// TIA Portal V19 export
ORGANIZATION_BLOCK "Main"   // OB3101, LAD, ProgramCycle
TITLE = "Main Program Sweep (Cycle)"
// stored: AutoNumber false, IsIECCheckEnabled true, Namespace Unit3.EM0, SetENOAutomatically true
   VAR_INPUT
      Initial_Call : Bool;   // Initial call of this OB
      Remanence : Bool;   // =True, if remanent data are available
   END_VAR
BEGIN

REGION Network 1 (SCL): Call Equipment
   "Unit3.EM0.CallEquipment_DB"(unitStatus := "Unit3.EmNodes".unitStatus,
                    unitAlarmDB := "Unit3.Alarms".emAlarms[Unit3_EM0],
                    emFeedback := "Unit3.EmNodes".emFeedback[Unit3_EM0]);
END_REGION
END_ORGANIZATION_BLOCK
